// TwinCAT 3 PLC project Demo
// ProgramVersion: 3.1.4022.3
// libraries:
//   Tc2_EtherCAT, * (Beckhoff Automation GmbH)
//   Tc2_SerialCom, * (Beckhoff Automation GmbH)
//   Tc2_Standard, * (Beckhoff Automation GmbH)
//   Tc2_System, * (Beckhoff Automation GmbH)
//   Tc2_Utilities, * (Beckhoff Automation GmbH)
//   Tc3_Module, * (Beckhoff Automation GmbH)
// project tree:
//   lcls-general/ FB_AnalogInput.TcPOU (not stored), FB_AnalogOutput.TcPOU (not stored), FB_BasicStats.TcPOU (not stored), FB_CoE_FastRead.TcPOU, FB_DataBuffer.TcPOU (not stored), FB_EL6_Com.TcPOU (not stored), FB_LREALBuffer.TcPOU (not stored), FB_ThermoCouple.TcPOU (not stored), FB_TimeStampBuffer.TcPOU (not stored), FB_TimeStampBufferGlobal.TcPOU (not stored), FB_UnixTimeStamp.TcPOU (not stored), FB_UnixTimeStampGlobal.TcPOU (not stored)
//   / PlcTask.TcTTO
//   POUs/ MAIN.TcPOU
// real-time tasks:
//   TASK PlcTask: cycle T#1ms, priority 20, ADS port 350
// motion (NC):
//   TASK NC-Task 1 SAF: cycle T#1ms, priority 4, ADS port 501
//   TASK NC-Task 1 SVB: cycle T#10ms, priority 8, ADS port 511
//   AXIS Axis 1 (id 1)
//     OtherSettings: AllowMotionCmdToSlave=true
//     encoder EncType=4
//       EncPara: MaxCount=#x0000ffff
//         Inc: RefSoftSyncMask=#x0000ffff
//     drive DrvType=24
//       Analog: ScaleFactorActTorque=0.1
//       TimeComp: TaskDelayCycles=1
//     controller CtrType=1
//       CtrPara: PriorControlFactor=1
//         Observer: BandWidth=20
//   AXIS Axis 2 (id 2)
//     OtherSettings: AllowMotionCmdToSlave=true
//     encoder EncType=4
//       EncPara: MaxCount=#x0000ffff
//         Inc: RefSoftSyncMask=#x0000ffff
//     drive DrvType=24
//       Analog: ScaleFactorActTorque=0.1
//       TimeComp: TaskDelayCycles=1
//     controller CtrType=1
//       CtrPara: PriorControlFactor=1
//         Observer: BandWidth=20
// I/O:
//   DEVICE Device 1 (EtherCAT), AmsNetId 172.21.42.227.2.1
//     Term 1 (EK1200) [EK1200-5000 EtherCAT Power supply (2A E-Bus)]
//       Term 2 (EL7041) [EL7041 1Ch. Stepper motor output stage (50V, 5A)]
//       Term 3 (EL5042) [EL5042 2Ch. BiSS-C Encoder]
//       Term 4 (EL7047) [EL7047 1Ch. Stepper motor output stage (50V, 5A)]
//       Term 5 (EL9011) [EL9011 End Terminal]
// variable links:
//   (this object) <-> Device 1 (EtherCAT)/Term 1 (EK1200)/Term 2 (EL7041)
//     Drive/Inputs/In/nState1 @bit 3 <-> STM Status/Status/Error
//     Drive/Inputs/In/nState1 @bit 5 <-> STM Status/Status/Moving negative
//     Drive/Inputs/In/nState1 @bit 4 <-> STM Status/Status/Moving positive
//     Drive/Inputs/In/nState1 @bit 1 <-> STM Status/Status/Ready
//     Drive/Inputs/In/nState1 <-> STM Status/Status/Ready to enable
//     Drive/Inputs/In/nState1 @bit 6 <-> STM Status/Status/Torque reduced
//     Drive/Inputs/In/nState1 @bit 2 <-> STM Status/Status/Warning
//     Drive/Inputs/In/nState2 @bit 3 <-> STM Status/Status/Digital input 1
//     Drive/Inputs/In/nState2 @bit 4 <-> STM Status/Status/Digital input 2
//     Drive/Inputs/In/nState2 @bit 5 <-> STM Status/Status/Sync error
//     Drive/Inputs/In/nState2 @bit 7 <-> STM Status/Status/TxPDO Toggle
//     Drive/Inputs/In/nState4 @bit 1 <-> WcState/InputToggle
//     Drive/Inputs/In/nState4 <-> WcState/WcState
//     Drive/Outputs/Out/nCtrl1 <-> STM Control/Control/Enable
//     Drive/Outputs/Out/nCtrl1 @bit 2 <-> STM Control/Control/Reduce torque
//     Drive/Outputs/Out/nCtrl1 @bit 1 <-> STM Control/Control/Reset
//     Drive/Outputs/Out/nDataOut2[0] <-> STM Velocity/Velocity
//     Enc/Inputs/In/nDataIn1[0] <-> ENC Status compact/Counter value
//     Enc/Inputs/In/nDataIn2[0] <-> ENC Status compact/Latch value
//     Enc/Inputs/In/nState1 @bit 4 <-> ENC Status compact/Status/Counter overflow
//     Enc/Inputs/In/nState1 @bit 3 <-> ENC Status compact/Status/Counter underflow
//     Enc/Inputs/In/nState1 @bit 7 <-> ENC Status compact/Status/Extrapolation stall
//     Enc/Inputs/In/nState1 <-> ENC Status compact/Status/Latch C valid
//     Enc/Inputs/In/nState1 @bit 1 <-> ENC Status compact/Status/Latch extern valid
//     Enc/Inputs/In/nState1 @bit 2 <-> ENC Status compact/Status/Set counter done
//     Enc/Inputs/In/nState2 @bit 4 <-> ENC Status compact/Status/Status of extern latch
//     Enc/Inputs/In/nState2 <-> ENC Status compact/Status/Status of input A
//     Enc/Inputs/In/nState2 @bit 1 <-> ENC Status compact/Status/Status of input B
//     Enc/Inputs/In/nState2 @bit 2 <-> ENC Status compact/Status/Status of input C
//     Enc/Inputs/In/nState2 @bit 5 <-> ENC Status compact/Status/Sync error
//     Enc/Inputs/In/nState2 @bit 7 <-> ENC Status compact/Status/TxPDO Toggle
//     Enc/Inputs/In/nState4 @bit 1 <-> WcState/InputToggle
//     Enc/Inputs/In/nState4 <-> WcState/WcState
//     Enc/Outputs/Out/nCtrl1 <-> ENC Control compact/Control/Enable latch C
//     Enc/Outputs/Out/nCtrl1 @bit 3 <-> ENC Control compact/Control/Enable latch extern on negative edge
//     Enc/Outputs/Out/nCtrl1 @bit 1 <-> ENC Control compact/Control/Enable latch extern on positive edge
//     Enc/Outputs/Out/nCtrl1 @bit 2 <-> ENC Control compact/Control/Set counter
//     Enc/Outputs/Out/nDataOut1[0] <-> ENC Control compact/Set counter value
//   (this object) <-> Device 1 (EtherCAT)/Term 1 (EK1200)/Term 4 (EL7047)
//     Drive/Inputs/In/nState1 @bit 3 <-> STM Status/Status/Error
//     Drive/Inputs/In/nState1 @bit 7 <-> STM Status/Status/Motor stall
//     Drive/Inputs/In/nState1 @bit 5 <-> STM Status/Status/Moving negative
//     Drive/Inputs/In/nState1 @bit 4 <-> STM Status/Status/Moving positive
//     Drive/Inputs/In/nState1 @bit 1 <-> STM Status/Status/Ready
//     Drive/Inputs/In/nState1 <-> STM Status/Status/Ready to enable
//     Drive/Inputs/In/nState1 @bit 6 <-> STM Status/Status/Torque reduced
//     Drive/Inputs/In/nState1 @bit 2 <-> STM Status/Status/Warning
//     Drive/Inputs/In/nState2 @bit 3 <-> STM Status/Status/Digital input 1
//     Drive/Inputs/In/nState2 @bit 4 <-> STM Status/Status/Digital input 2
//     Drive/Inputs/In/nState2 @bit 5 <-> STM Status/Status/Sync error
//     Drive/Inputs/In/nState2 @bit 7 <-> STM Status/Status/TxPDO Toggle
//     Drive/Inputs/In/nState4 @bit 1 <-> WcState/InputToggle
//     Drive/Inputs/In/nState4 <-> WcState/WcState
//     Drive/Outputs/Out/nCtrl1 <-> STM Control/Control/Enable
//     Drive/Outputs/Out/nCtrl1 @bit 2 <-> STM Control/Control/Reduce torque
//     Drive/Outputs/Out/nCtrl1 @bit 1 <-> STM Control/Control/Reset
//     Drive/Outputs/Out/nCtrl2 @bit 3 <-> STM Control/Control/Digital output 1
//     Drive/Outputs/Out/nDataOut2[0] <-> STM Velocity/Velocity
//     Enc/Inputs/In/nDataIn1[0] <-> ENC Status compact/Counter value
//     Enc/Inputs/In/nDataIn2[0] <-> ENC Status compact/Latch value
//     Enc/Inputs/In/nState1 @bit 4 <-> ENC Status compact/Status/Counter overflow
//     Enc/Inputs/In/nState1 @bit 3 <-> ENC Status compact/Status/Counter underflow
//     Enc/Inputs/In/nState1 @bit 7 <-> ENC Status compact/Status/Extrapolation stall
//     Enc/Inputs/In/nState1 <-> ENC Status compact/Status/Latch C valid
//     Enc/Inputs/In/nState1 @bit 1 <-> ENC Status compact/Status/Latch extern valid
//     Enc/Inputs/In/nState1 @bit 2 <-> ENC Status compact/Status/Set counter done
//     Enc/Inputs/In/nState2 @bit 4 <-> ENC Status compact/Status/Status of extern latch
//     Enc/Inputs/In/nState2 <-> ENC Status compact/Status/Status of input A
//     Enc/Inputs/In/nState2 @bit 1 <-> ENC Status compact/Status/Status of input B
//     Enc/Inputs/In/nState2 @bit 2 <-> ENC Status compact/Status/Status of input C
//     Enc/Inputs/In/nState2 @bit 5 <-> ENC Status compact/Status/Sync error
//     Enc/Inputs/In/nState2 @bit 7 <-> ENC Status compact/Status/TxPDO Toggle
//     Enc/Inputs/In/nState4 @bit 1 <-> WcState/InputToggle
//     Enc/Inputs/In/nState4 <-> WcState/WcState
//     Enc/Outputs/Out/nCtrl1 <-> ENC Control compact/Control/Enable latch C
//     Enc/Outputs/Out/nCtrl1 @bit 3 <-> ENC Control compact/Control/Enable latch extern on negative edge
//     Enc/Outputs/Out/nCtrl1 @bit 1 <-> ENC Control compact/Control/Enable latch extern on positive edge
//     Enc/Outputs/Out/nCtrl1 @bit 2 <-> ENC Control compact/Control/Set counter
//     Enc/Outputs/Out/nDataOut1[0] <-> ENC Control compact/Set counter value
//   Demo Instance <-> Device 1 (EtherCAT)/Term 1 (EK1200)/Term 2 (EL7041)
//     PlcTask Inputs/MAIN.fbCoEFast.stPlcDriveRef/aNetId <-> InfoData/AdsAddr/netId
//     PlcTask Inputs/MAIN.fbCoEFast.stPlcDriveRef/nSlaveAddr <-> InfoData/AdsAddr/port

CONFIGURATION Demo
    RESOURCE PLC ON TwinCAT3
        TASK PlcTask(INTERVAL := T#1ms, PRIORITY := 20);
        PROGRAM MAIN WITH PlcTask : MAIN;
    END_RESOURCE
END_CONFIGURATION

// ---- POUs/MAIN.TcPOU
PROGRAM MAIN
VAR
	fbCoEFast: FB_CoE_FastRead;
	fbData: FB_LREALBuffer;
	fbTime: FB_TimeStampBuffer;
	fbStats: FB_BasicStats;
	fbAO: FB_AnalogOutput;
	fbAI: FB_AnalogInput;
	
	fbTC: FB_ThermoCouple;
	fbSer: FB_EL6_Com;

	rng: DRAND;
	fVoltOut: LREAL;
	fVoltIn: LREAL;
	nTermOut AT %Q*: INT;
	iTermIn AT %I*: INT;
	
	fCoilA: INT;
END_VAR

fbCoEFast(
	bExecute := TRUE,
	nIndex := 16#9010,
	nSubIndex := 16#04,
	pDstBuf := ADR(fCoilA),
	cbBufLen := SIZEOF(fCoilA));

fbData(
	bExecute := rng.Num > 0.5,
	fInput := fCoilA);

fbTime(
	bExecute := rng.Num > 0.5);

fbStats(
	aSignal := fbData.arrOutput,
	bExecute := fbData.bNewArray);

fbAO(
	fReal := fVoltOut, // Volts
	fSafeMax := 8, // Volts
	fSafeMin := 0, // Volts
	iTermBits := 16, // Bits
	fTermMax := 10, // Volts
	fTermMin := 0, // Volts
	iRaw => nTermOut); // 16 bit integer

fbAI(
	iRaw := iTermIn, // 16 bit integer
	iTermBits := 16, // Bits
	fTermMax := 10, // Volts
	fTermMin := -10, // Volts
	fReal => fVoltIn); // Volts

rng();

END_PROGRAM

// ---- lcls-general/FB_CoE_FastRead.TcPOU
FUNCTION_BLOCK FB_CoE_FastRead
(*
	Utility to repeatedly read a CoE parameter
	2019-10-09 Zachary Lentz
	
	In practice, it's impossible to read most CoE parameters every cycle,
	but this is a best effort and will work if the data is available
*)
VAR_INPUT
	// If TRUE we'll attempt a CoE read this cycle.
	bExecute: BOOL;
	// Link this to your terminal's drive reference variables under InfoData.
	stPlcDriveRef AT %I*: ST_PlcDriveRef;
	// Hexadecimal index of CoE, e.g. the 8010 in 8010:12
	nIndex: UINT;
	// Hexadecimal subindex of CoE, e.g. the 12 in 8010:12
	nSubIndex: BYTE;
	// Pointer to a value to fill with the result of the read, e.g. ADR(MyValue)
	pDstBuf: PVOID;
	// Data size of pDstBuf, e.g. SIZEOF(MyValue)
	cbBufLen: UINT;
END_VAR
VAR_OUTPUT
	// TRUE if the value was updated on this cycle.
	bNewValue: BOOL;
END_VAR
VAR
	fbRead: FB_CoERead_ByDriveRef;
	stDriveRef: ST_DriveRef;
	iLoop: INT;
	bInnerExec: BOOL;
END_VAR

stDriveRef.sNetId := F_CreateAmsNetId(stPlcDriveRef.aNetId);
stDriveRef.nSlaveAddr := stPlcDriveRef.nSlaveAddr;
stDriveRef.nDriveNo := stPlcDriveRef.nDriveNo;
stDriveRef.nDriveType := stPlcDriveRef.nDriveType;

bNewValue := FALSE;
IF bExecute THEN
	// You need to do this block 3 times per cycle to have a chance at always getting a read
	FOR iLoop:= 1 TO 3 DO
		fbRead(
			stDriveRef := stDriveRef,
			nIndex := nIndex,
			nSubIndex := nSubIndex,
			pDstBuf := pDstBuf,
			cbBufLen := cbBufLen,
			bExecute := bInnerExec,
			tTimeout := T#1s);
			
		IF bInnerExec AND NOT fbRead.bBusy AND NOT fbRead.bError THEN
			bInnerExec := FALSE;
			bNewValue := TRUE;
		ELSE
			bInnerExec := TRUE;
		END_IF
	END_FOR
END_IF

END_FUNCTION_BLOCK
